{attribute 'call_after_init'}
FUNCTION_BLOCK FB_Arbiter_Test EXTENDS FB_TestSuite IMPLEMENTS I_RunnableTestSuite
VAR_INPUT
END_VAR
VAR_OUTPUT
END_VAR
VAR
	fbAssert : TcUnit.FB_Assert;
END_VAR

METHOD PRIVATE Arbitration
VAR_INPUT
END_VAR
VAR
	fbArbiter	:	FB_Arbiter;
	
 	nAttReqID	:	UDINT	:= 1;
	stAttReqBP	:	ST_BeamParams := PMPS_GVL_BeamParams.cstFullBeam;
	
	nPPEReqID	:	UDINT	:= 2;
	stPPEReqBP	:	ST_BeamParams := PMPS_GVL_BeamParams.cstFullBeam;
	
	nEVReqID	:	UDINT	:= 3;
	stEVReqBP	:	ST_BeamParams := PMPS_GVL_BeamParams.cstFullBeam;
	
	nRateReqID	:	UDINT	:= 4;
	stRateReqBP	:	ST_BeamParams := PMPS_GVL_BeamParams.cstFullBeam;
	
	stArbitratedBP	:	ST_ReqBeamParams;
	stExpectedBP	:	ST_ReqBeamParams;
END_VAR
TEST('Arbitration');

//Initialize arbiter
fbArbiter.A_Init();

stAttReqBP.fAtt := 50;
stPPEReqBP.fPP_mJ := 1;
stEVReqBP.neVReqRange := 2#1111_1100_1111_1111;
stRateReqBP.nRate := 120;

//Load arbiter with beam parameter sets
fbAssert.AssertTrue(fbArbiter.AddRequest(nAttReqID, stAttReqBP),
					'Safest attenuation request failed to load');
					
//Load arbiter with beam parameter sets
fbAssert.AssertTrue(fbArbiter.AddRequest(nPPEReqID, stPPEReqBP),
					'Safest PPE request failed to load');
					
//Load arbiter with beam parameter sets
fbAssert.AssertTrue(fbArbiter.AddRequest(nEVReqID, stEVReqBP),
					'Safest stEVReqBP request failed to load');
					
//Load arbiter with beam parameter sets
fbAssert.AssertTrue(fbArbiter.AddRequest(nRateReqID, stRateReqBP),
					'Safest stEVReqBP request failed to load');

stExpectedBP.fAtt 	:= 	stAttReqBP.fAtt;
stExpectedBP.fPP_mJ	:=  stPPEReqBP.fPP_mJ;
stExpectedBP.neVPermRange := stEVReqBP.neVReqRange;
stExpectedBP.nRate := stRateReqBP.nRate;

stArbitratedBP := fbArbiter.GetArbitratedBP();

fbAssert.AssertFalse(F_DiffReqBeamParams(stExpectedBP, stArbitratedBP),
				'Arbitrated BP does not match expected.');
END_METHOD

METHOD FB_init : BOOL
VAR_INPUT
	bInitRetains : BOOL; // if TRUE, the retain variables are initialized (warm start / cold start)
	bInCopyCode : BOOL;  // if TRUE, the instance afterwards gets moved into the copy code (online change)
END_VAR
SUPER^.RegisterTestSuite(THIS^);
END_METHOD

METHOD PRIVATE RequestCheckRemoveBP
VAR_INPUT
END_VAR
VAR
	fbArbiter	:	FB_Arbiter;
	
	nId	:	DWORD := 1;
	stReq	:	ST_BeamParams;
END_VAR
fbArbiter.A_Init();

TEST('RequestBP');
fbAssert.AssertTrue(fbArbiter.AddRequest(nId, stReq),
	'Request failed');
	
TEST('DuplicateID');
fbAssert.AssertFalse(fbArbiter.AddRequest(nId, stReq),
	'Duplicate request accepted, not good.');
	
TEST('CheckBP');
fbAssert.AssertTrue(fbArbiter.CheckRequest(nId),
	'Check failed');
	
TEST('IDDoesNotExist');
fbAssert.AssertFalse(fbArbiter.CheckRequest(nId+1),
	'Check returned true when ID does not exist');
	
TEST('RemoveBP');
fbAssert.AssertTrue(fbArbiter.RemoveRequest(nId),
	'Remove failed');
fbAssert.AssertFalse(fbArbiter.CheckRequest(nId),
	'Remove did not remove request');
END_METHOD

METHOD RunTests : TCUNIT.E_TestSuiteRunState
Arbitration();
RequestCheckRemoveBP();

RunTests := TcUnit.E_TestSuiteRunState.FINISHED;
END_METHOD

END_FUNCTION_BLOCK

(* stored: Version 1.1.0.1, ProductVersion 3.1.4022.18
   POU FB_Arbiter_Test: Id {db09e55a-38f4-0816-2f75-9c1afd6ec43c}, SpecialFunc None
   Method Arbitration: Id {2b6f199f-ca1a-03e4-0a23-e2d3f0dbc445}
   Method FB_init: Id {905e10b5-34d1-0d47-0f2f-058acb702e66}
   Method RequestCheckRemoveBP: Id {8a012cde-0038-03e6-02ee-15f6a358c4a9}
   Method RunTests: Id {1d17ac00-7099-0d59-00bd-5e8356ee15d5} *)
